// TIA Portal V20 export
FUNCTION "右顶升伺服" : Void   // FC2, LAD
{ S7_Optimized_Access := 'TRUE' }
// stored: SetENOAutomatically false
BEGIN

REGION Network 1 (SCL)
   "右顶升V90控制字".%X0 := "1200_下载".位9;
   "右顶升V90控制字".%X1 := "1200_下载".位10;
   "右顶升V90控制字".%X2 := "1200_下载".位11;
   "右顶升V90控制字".%X3 := "1200_下载".位12;
   "右顶升V90控制字".%X4 := "1200_下载".位13;
   "右顶升V90控制字".%X5 := "1200_下载".位14;
   "右顶升V90控制字".%X6 := "1200_下载".位15;
   "右顶升V90控制字".%X7 := "1200_下载".位16;

   "右_回原模式" := "1200_下载".整型2;

   "右_绝对位置" := "1200_下载".浮点数6;
   "右_绝对速度" := "1200_下载".浮点数7;
   "右_相对位置" := "1200_下载".浮点数8;
   "右_相对速度" := "1200_下载".浮点数9;
   "右_点动速度" := "1200_下载".浮点数10;
END_REGION

REGION Network 2
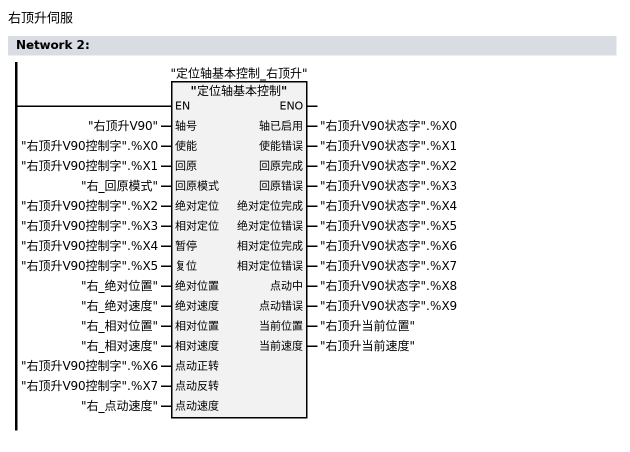
   RUNG wire#powerrail
      "定位轴基本控制_右顶升"(轴号 := "右顶升V90", 使能 := "右顶升V90控制字".%X0, 回原 := "右顶升V90控制字".%X1, 回原模式 := "右_回原模式", 绝对定位 := "右顶升V90控制字".%X2, 相对定位 := "右顶升V90控制字".%X3, 暂停 := "右顶升V90控制字".%X4, 复位 := "右顶升V90控制字".%X5, 绝对位置 := "右_绝对位置", 绝对速度 := "右_绝对速度", 相对位置 := "右_相对位置", 相对速度 := "右_相对速度", 点动正转 := "右顶升V90控制字".%X6, 点动反转 := "右顶升V90控制字".%X7, 点动速度 := "右_点动速度", 轴已启用 => "右顶升V90状态字".%X0, 使能错误 => "右顶升V90状态字".%X1, 回原完成 => "右顶升V90状态字".%X2, 回原错误 => "右顶升V90状态字".%X3, 绝对定位完成 => "右顶升V90状态字".%X4, 绝对定位错误 => "右顶升V90状态字".%X5, 相对定位完成 => "右顶升V90状态字".%X6, 相对定位错误 => "右顶升V90状态字".%X7, 点动中 => "右顶升V90状态字".%X8, 点动错误 => "右顶升V90状态字".%X9, 当前位置 => "右顶升当前位置", 当前速度 => "右顶升当前速度")
   END_RUNG
   // the same network as SCL:
   "定位轴基本控制_右顶升"(轴号 := "右顶升V90",   // "定位轴基本控制"
                 使能 := "右顶升V90控制字".%X0,
                 回原 := "右顶升V90控制字".%X1,
                 回原模式 := "右_回原模式",
                 绝对定位 := "右顶升V90控制字".%X2,
                 相对定位 := "右顶升V90控制字".%X3,
                 暂停 := "右顶升V90控制字".%X4,
                 复位 := "右顶升V90控制字".%X5,
                 绝对位置 := "右_绝对位置",
                 绝对速度 := "右_绝对速度",
                 相对位置 := "右_相对位置",
                 相对速度 := "右_相对速度",
                 点动正转 := "右顶升V90控制字".%X6,
                 点动反转 := "右顶升V90控制字".%X7,
                 点动速度 := "右_点动速度",
                 轴已启用 => "右顶升V90状态字".%X0,
                 使能错误 => "右顶升V90状态字".%X1,
                 回原完成 => "右顶升V90状态字".%X2,
                 回原错误 => "右顶升V90状态字".%X3,
                 绝对定位完成 => "右顶升V90状态字".%X4,
                 绝对定位错误 => "右顶升V90状态字".%X5,
                 相对定位完成 => "右顶升V90状态字".%X6,
                 相对定位错误 => "右顶升V90状态字".%X7,
                 点动中 => "右顶升V90状态字".%X8,
                 点动错误 => "右顶升V90状态字".%X9,
                 当前位置 => "右顶升当前位置",
                 当前速度 => "右顶升当前速度");
END_REGION

REGION Network 3 (SCL)
   "1200_上传".位11 := "右顶升V90状态字".%X0;
   "1200_上传".位12 := "右顶升V90状态字".%X1;
   "1200_上传".位13 := "右顶升V90状态字".%X2;
   "1200_上传".位14 := "右顶升V90状态字".%X3;
   "1200_上传".位15 := "右顶升V90状态字".%X4;
   "1200_上传".位16 := "右顶升V90状态字".%X5;
   "1200_上传".位17 := "右顶升V90状态字".%X6;
   "1200_上传".位18 := "右顶升V90状态字".%X7;
   "1200_上传".位19 := "右顶升V90状态字".%X8;
   "1200_上传".位20 := "右顶升V90状态字".%X9;

   "1200_上传".浮点数3 := "右顶升当前位置";
   "1200_上传".浮点数4 := "右顶升当前速度";
END_REGION
END_FUNCTION
